{attribute 'linkalways'} 
{attribute 'no_explicit_call' := 'This FB is a CLASS and must be accessed using methods or properties'}
{attribute 'enable_dynamic_creation'}
FUNCTION_BLOCK EventGroupItem EXTENDS Disposable IMPLEMENTS I_EventGroupItem
VAR
	name : T_MAXSTRING;
	firstEventHandlerItem : I_EventHandlerItem;
	_next : I_EventGroupItem;
	_previous : I_EventGroupItem;
END_VAR

METHOD PUBLIC AddHandler
VAR_INPUT
	EventHandler : I_EventHandler;
END_VAR
AddNewEventHandlerItem(EventHandler);
END_METHOD

METHOD PUBLIC AddNewEventHandlerItem : I_EventHandlerItem
VAR_INPUT
	EventHandler : I_EventHandler;
END_VAR
VAR
	pEventHandlerItem : POINTER TO EventHandlerItem;
END_VAR
pEventHandlerItem := __NEW(EventHandlerItem(Handler := EventHandler));
InsertEventHandlerItem(pEventHandlerItem^);
AddNewEventHandlerItem := pEventHandlerItem^;
END_METHOD

METHOD PUBLIC Emit
VAR_INPUT
	Event : I_Event;
END_VAR
VAR
	currentEventHandlerItem : I_EventHandlerItem;
END_VAR
currentEventHandlerItem := firstEventHandlerItem;

WHILE currentEventHandlerItem <> 0 DO
	currentEventHandlerItem.Emit(Event);
	currentEventHandlerItem := currentEventHandlerItem.Next;
END_WHILE
END_METHOD

METHOD EqualTo : BOOL
VAR_INPUT
	Name : T_MAXSTRING;
END_VAR
EqualTo := THIS^.name = Name;
END_METHOD

METHOD FB_init : BOOL
VAR_INPUT
	bInitRetains : BOOL; // if TRUE, the retain variables are initialized (warm start / cold start)
	bInCopyCode : BOOL;  // if TRUE, the instance afterwards gets moved into the copy code (online change)
	GroupName : T_MAXSTRING;
END_VAR
name := GroupName;
END_METHOD

METHOD PRIVATE FindEventHandlerItemByHandler : I_EventHandlerItem
VAR_INPUT
	EventHandler : I_EventHandler;
END_VAR
VAR
	currentEventHandlerItem : I_EventHandlerItem;
END_VAR
currentEventHandlerItem := firstEventHandlerItem;

WHILE currentEventHandlerItem <> 0 DO
	
	IF currentEventHandlerItem.EqualTo(EventHandler) THEN
		FindEventHandlerItemByHandler := currentEventHandlerItem; 
		RETURN;
	END_IF
	
	currentEventHandlerItem := currentEventHandlerItem.Next;

END_WHILE
END_METHOD

PROPERTY HasHandlers : BOOL
GET
HasHandlers := firstEventHandlerItem <> 0;
END_GET
END_PROPERTY

METHOD PRIVATE InsertEventHandlerItem
VAR_INPUT
	EventHandlerItem : I_EventHandlerItem;
END_VAR
VAR
	currentEventHandlerItem : I_EventHandlerItem;
END_VAR
IF firstEventHandlerItem = 0 THEN
	firstEventHandlerItem := EventHandlerItem;
	RETURN;
END_IF

currentEventHandlerItem := firstEventHandlerItem;

WHILE currentEventHandlerItem.next <> 0 DO
	currentEventHandlerItem := currentEventHandlerItem.next;
END_WHILE

currentEventHandlerItem.next := EventHandlerItem;
EventHandlerItem.previous := currentEventHandlerItem;
END_METHOD

PROPERTY PUBLIC Next : I_EventGroupItem
GET
Next := _next;
END_GET
SET
_next := Next;
END_SET
END_PROPERTY

METHOD PROTECTED OnDispose : BOOL
VAR_INPUT
	CalledExplicitly : BOOL;
END_VAR
RemoveAllEventHandlerItems();
END_METHOD

PROPERTY PUBLIC Previous : I_EventGroupItem
GET
Previous := _previous;
END_GET
SET
_previous := Previous;
END_SET
END_PROPERTY

METHOD PRIVATE RemoveAllEventHandlerItems
VAR_INPUT
END_VAR
WHILE firstEventHandlerItem <> 0 DO
	RemoveEventHandlerItem(firstEventHandlerItem);
END_WHILE
END_METHOD

METHOD PRIVATE RemoveEventHandlerItem
VAR_INPUT
	EventHandlerItem : I_EventHandlerItem;
END_VAR
RemoveEventHandlerItemFromCollection(EventHandlerItem);
EventHandlerItem.Dispose();
END_METHOD

METHOD PRIVATE RemoveEventHandlerItemFromCollection
VAR_INPUT
	EventHandlerItem : I_EventHandlerItem;
END_VAR
VAR
	previous : I_EventHandlerItem;
	next : I_EventHandlerItem;
END_VAR
IF EventHandlerItem = 0 THEN
	// nothing to remove
	RETURN;
END_IF

IF EventHandlerItem = firstEventHandlerItem AND EventHandlerItem.Next = 0 THEN 
	
	// the item was the only one in the list, as such you just set the first to zero
	firstEventHandlerItem := 0; 
	
ELSIF EventHandlerItem = firstEventHandlerItem THEN 
	
	// the item was the first in the list of many, so make the next item the first and remove 
	// it's "previous" as the first in the item does not have a previous
	firstEventHandlerItem := EventHandlerItem.next; 
	firstEventHandlerItem.Previous := 0;

ELSIF EventHandlerItem.Next <> 0 THEN
	
	// the item is mid list so link it's previous and next together 
	previous := EventHandlerItem.Previous;
	next := EventHandlerItem.Next;
	
	previous.Next := next;
	next.Previous := previous;
	
ELSE 
	
	// the item is at the end so only remove itself from the previous
	previous := EventHandlerItem.Previous;
	previous.Next := 0;

END_IF
END_METHOD

METHOD RemoveHandler
VAR_INPUT
	EventHandler : I_EventHandler;
END_VAR
VAR
	foundHandlerItem : I_EventHandlerItem;
END_VAR
foundHandlerItem := FindEventHandlerItemByHandler(EventHandler);

IF foundHandlerItem = 0 THEN
	RETURN;
END_IF

RemoveEventHandlerItem(foundHandlerItem);
END_METHOD

END_FUNCTION_BLOCK

(* stored: Version 1.1.0.1, ProductVersion 3.1.4024.12
   POU EventGroupItem: Id {64482246-e111-09c5-0503-b887468d0fba}, SpecialFunc None
   Folder Constructor: Id {6b4faf6d-908a-0f96-192d-76e2be6cc1f1}
   Folder Private: Id {c1622086-a143-03da-206d-9fe068b400ff}
   Folder Protected: Id {bd343c31-90dd-4403-8dd5-e3eb56fb246f}
   Method AddHandler: Id {997b0bc9-2d2d-03f8-228b-b62bbd3eb317}
   Method AddNewEventHandlerItem: Id {5362dc37-d444-0f4e-2f81-e06b34fc0e73}
   Method Emit: Id {e60b34f8-9fa7-0f6b-2b74-93fdf67e7f67}
   Method EqualTo: Id {328d40f5-e3c2-0cda-1f3d-eed7bb83e6a8}
   Method FB_init: Id {f87ac4b2-1713-052a-21e8-dd9974477c00}
   Method FindEventHandlerItemByHandler: Id {5be8512f-8916-066a-0ade-3f4977175730}
   Property HasHandlers: Id {e0ca0a53-c8d7-0021-1c9e-45e1453cb912}
   Get Get: Id {bb253f2e-09a0-07b1-26ca-7d38f485fe9a}
   Method InsertEventHandlerItem: Id {79d70cb5-7a1c-0779-0ab4-d1fb73717a1c}
   Property Next: Id {6bd16881-506e-0380-18bb-934857c46061}
   Get Get: Id {235b1fc8-fd04-05be-2dd9-19b75bfcde09}
   Set Set: Id {f6e0cc02-b082-0ea7-3f8b-fa9fd5da610d}
   Method OnDispose: Id {12515b58-aff7-4c18-b080-92c582058756}
   Property Previous: Id {05aac4f6-018a-0924-2c76-20ad77628642}
   Get Get: Id {f35de5bb-2f2a-0177-28ee-f5f82b6c3802}
   Set Set: Id {e87f3474-fe0c-0306-15ea-e351409dc278}
   Method RemoveAllEventHandlerItems: Id {22db252f-5d74-4769-8122-f4dda925b209}
   Method RemoveEventHandlerItem: Id {f97a2596-68d2-0ec3-0c71-2d8f13ace3bb}
   Method RemoveEventHandlerItemFromCollection: Id {8e960e12-b617-0e73-0998-bc0951492a6d}
   Method RemoveHandler: Id {53bbcc04-313f-0ca5-1c3a-a1d00218bc46} *)
